(* CODESYS project FU_dwBitGet.xml

Project tree, tasks and I/O mapping:
  function FU_dwBitGet [ST]
*)

// FU_dwBitGet
//This function get the bit value from a variable
// |**Version**|**Author**| **Date** |**Changes**
// | 1         | NSN      | 11-01-19 | Creation
FUNCTION FU_dwBitGet : BOOL
VAR_INPUT
	dbVar	:DWORD;		//The value to work with
	bIndex	:BYTE;		//Which bit to get	
END_VAR

FU_dwBitGet		:=		(dbVar AND SHL(1,bIndex)) <> 0;

END_FUNCTION
